   1:  PR[GP1:91,1] = PR[GP1:90,1] + 14.958;
   1:  PR[GP1:91,2] = PR[GP1:90,2] + 47.026;
   1:L PR[91] R[100]mm/sec CNT100;
   1:  PR[GP1:91,1] = PR[GP1:90,1] + 1.682;
   1:  PR[GP1:91,2] = PR[GP1:90,2] + 49.128;
   1:L PR[91] R[100]mm/sec CNT100;
   1:  PR[GP1:91,1] = PR[GP1:90,1] + 0.106;
   1:  PR[GP1:91,2] = PR[GP1:90,2] + 49.323;
   1:L PR[91] R[100]mm/sec CNT100;
   1:  ! -- Layer/Ebene 225 -- !;
   1:  PR[91] = PR[90];
   1:  PR[GP1:91,1] = PR[GP1:90,1] + -0.725;
   1:  PR[GP1:91,2] = PR[GP1:90,2] + 49.220;
   1:  PR[GP1:91,3] = PR[GP1:90,3] + 137.555;
   1:L PR[91] R[100]mm/sec CNT100;
   1:  PR[GP1:91,1] = PR[GP1:90,1] + -14.943;
   1:  PR[GP1:91,2] = PR[GP1:90,2] + 46.968;
   1:L PR[91] R[100]mm/sec CNT100;
   1:  PR[GP1:91,1] = PR[GP1:90,1] + -15.715;
   1:  PR[GP1:91,2] = PR[GP1:90,2] + 46.669;
   1:L PR[91] R[100]mm/sec CNT100;
   1:  PR[GP1:91,1] = PR[GP1:90,1] + -28.542;
   1:  PR[GP1:91,2] = PR[GP1:90,2] + 40.134;
   1:L PR[91] R[100]mm/sec CNT100;
   1:  PR[GP1:91,1] = PR[GP1:90,1] + -29.217;
   1:  PR[GP1:91,2] = PR[GP1:90,2] + 39.656;
   1:L PR[91] R[100]mm/sec CNT100;
   1:  PR[GP1:91,1] = PR[GP1:90,1] + -39.393;
   1:  PR[GP1:91,2] = PR[GP1:90,2] + 29.479;
   1:L PR[91] R[100]mm/sec CNT100;
   1:  PR[GP1:91,1] = PR[GP1:90,1] + -39.995;
   1:  PR[GP1:91,2] = PR[GP1:90,2] + 28.755;
   1:L PR[91] R[100]mm/sec CNT100;
   1:  PR[GP1:91,1] = PR[GP1:90,1] + -46.526;
   1:  PR[GP1:91,2] = PR[GP1:90,2] + 15.936;
   1:L PR[91] R[100]mm/sec CNT100;
   1:  PR[GP1:91,1] = PR[GP1:90,1] + -46.904;
   1:  PR[GP1:91,2] = PR[GP1:90,2] + 15.080;
   1:L PR[91] R[100]mm/sec CNT100;
   1:  PR[GP1:91,1] = PR[GP1:90,1] + -47.036;
   1:  PR[GP1:91,2] = PR[GP1:90,2] + 14.132;
   1:L PR[91] R[100]mm/sec CNT100;
   1:  PR[GP1:91,1] = PR[GP1:90,1] + -49.287;
   1:  PR[GP1:91,2] = PR[GP1:90,2] + -0.078;
   1:L PR[91] R[100]mm/sec CNT100;
   1:  PR[GP1:91,1] = PR[GP1:90,1] + -49.157;
   1:  PR[GP1:91,2] = PR[GP1:90,2] + -1.010;
   1:L PR[91] R[100]mm/sec CNT100;
   1:  PR[GP1:91,1] = PR[GP1:90,1] + -46.906;
   1:  PR[GP1:91,2] = PR[GP1:90,2] + -15.219;
   1:L PR[91] R[100]mm/sec CNT100;
   1:  PR[GP1:91,1] = PR[GP1:90,1] + -46.526;
   1:  PR[GP1:91,2] = PR[GP1:90,2] + -16.080;
   1:L PR[91] R[100]mm/sec CNT100;
   1:  PR[GP1:91,1] = PR[GP1:90,1] + -39.995;
   1:  PR[GP1:91,2] = PR[GP1:90,2] + -28.899;
   1:L PR[91] R[100]mm/sec CNT100;
   1:  PR[GP1:91,1] = PR[GP1:90,1] + -39.393;
   1:  PR[GP1:91,2] = PR[GP1:90,2] + -29.623;
   1:L PR[91] R[100]mm/sec CNT100;
   1:  PR[GP1:91,1] = PR[GP1:90,1] + -29.217;
   1:  PR[GP1:91,2] = PR[GP1:90,2] + -39.800;
   1:L PR[91] R[100]mm/sec CNT100;
   1:  PR[GP1:91,1] = PR[GP1:90,1] + -28.542;
   1:  PR[GP1:91,2] = PR[GP1:90,2] + -40.278;
   1:L PR[91] R[100]mm/sec CNT100;
   1:  PR[GP1:91,1] = PR[GP1:90,1] + -15.715;
   1:  PR[GP1:91,2] = PR[GP1:90,2] + -46.813;
   1:L PR[91] R[100]mm/sec CNT100;
   1:  PR[GP1:91,1] = PR[GP1:90,1] + -14.953;
   1:  PR[GP1:91,2] = PR[GP1:90,2] + -47.109;
   1:L PR[91] R[100]mm/sec CNT100;
   1:  PR[GP1:91,1] = PR[GP1:90,1] + -14.102;
   1:  PR[GP1:91,2] = PR[GP1:90,2] + -47.214;
   1:L PR[91] R[100]mm/sec CNT100;
   1:  PR[GP1:91,1] = PR[GP1:90,1] + 0.117;
   1:  PR[GP1:91,2] = PR[GP1:90,2] + -49.466;
   1:L PR[91] R[100]mm/sec CNT100;
   1:  PR[GP1:91,1] = PR[GP1:90,1] + 0.938;
   1:  PR[GP1:91,2] = PR[GP1:90,2] + -49.364;
   1:L PR[91] R[100]mm/sec CNT100;
   1:  PR[GP1:91,1] = PR[GP1:90,1] + 15.156;
   1:  PR[GP1:91,2] = PR[GP1:90,2] + -47.112;
   1:L PR[91] R[100]mm/sec CNT100;
   1:  PR[GP1:91,1] = PR[GP1:90,1] + 15.928;
   1:  PR[GP1:91,2] = PR[GP1:90,2] + -46.813;
   1:L PR[91] R[100]mm/sec CNT100;
   1:  PR[GP1:91,1] = PR[GP1:90,1] + 28.755;
   1:  PR[GP1:91,2] = PR[GP1:90,2] + -40.278;
   1:L PR[91] R[100]mm/sec CNT100;
   1:  PR[GP1:91,1] = PR[GP1:90,1] + 29.430;
   1:  PR[GP1:91,2] = PR[GP1:90,2] + -39.800;
   1:L PR[91] R[100]mm/sec CNT100;
   1:  PR[GP1:91,1] = PR[GP1:90,1] + 39.607;
   1:  PR[GP1:91,2] = PR[GP1:90,2] + -29.623;
   1:L PR[91] R[100]mm/sec CNT100;
   1:  PR[GP1:91,1] = PR[GP1:90,1] + 40.208;
   1:  PR[GP1:91,2] = PR[GP1:90,2] + -28.899;
   1:L PR[91] R[100]mm/sec CNT100;
   1:  PR[GP1:91,1] = PR[GP1:90,1] + 46.739;
   1:  PR[GP1:91,2] = PR[GP1:90,2] + -16.080;
   1:L PR[91] R[100]mm/sec CNT100;
   1:  PR[GP1:91,1] = PR[GP1:90,1] + 47.117;
   1:  PR[GP1:91,2] = PR[GP1:90,2] + -15.224;
   1:L PR[91] R[100]mm/sec CNT100;
   1:  PR[GP1:91,1] = PR[GP1:90,1] + 47.250;
   1:  PR[GP1:91,2] = PR[GP1:90,2] + -14.275;
   1:L PR[91] R[100]mm/sec CNT100;
   1:  PR[GP1:91,1] = PR[GP1:90,1] + 49.500;
   1:  PR[GP1:91,2] = PR[GP1:90,2] + -0.066;
   1:L PR[91] R[100]mm/sec CNT100;
   1:  PR[GP1:91,1] = PR[GP1:90,1] + 49.370;
   1:  PR[GP1:91,2] = PR[GP1:90,2] + 0.866;
   1:L PR[91] R[100]mm/sec CNT100;
   1:  PR[GP1:91,1] = PR[GP1:90,1] + 47.119;
   1:  PR[GP1:91,2] = PR[GP1:90,2] + 15.075;
   1:L PR[91] R[100]mm/sec CNT100;
   1:  PR[GP1:91,1] = PR[GP1:90,1] + 46.739;
   1:  PR[GP1:91,2] = PR[GP1:90,2] + 15.936;
   1:L PR[91] R[100]mm/sec CNT100;
   1:  PR[GP1:91,1] = PR[GP1:90,1] + 40.208;
   1:  PR[GP1:91,2] = PR[GP1:90,2] + 28.755;
   1:L PR[91] R[100]mm/sec CNT100;
   1:  PR[GP1:91,1] = PR[GP1:90,1] + 39.607;
   1:  PR[GP1:91,2] = PR[GP1:90,2] + 29.479;
   1:L PR[91] R[100]mm/sec CNT100;
   1:  PR[GP1:91,1] = PR[GP1:90,1] + 29.430;
   1:  PR[GP1:91,2] = PR[GP1:90,2] + 39.656;
   1:L PR[91] R[100]mm/sec CNT100;
   1:  PR[GP1:91,1] = PR[GP1:90,1] + 28.755;
   1:  PR[GP1:91,2] = PR[GP1:90,2] + 40.134;
   1:L PR[91] R[100]mm/sec CNT100;
   1:  PR[GP1:91,1] = PR[GP1:90,1] + 15.928;
   1:  PR[GP1:91,2] = PR[GP1:90,2] + 46.669;
   1:L PR[91] R[100]mm/sec CNT100;
   1:  PR[GP1:91,1] = PR[GP1:90,1] + 15.156;
   1:  PR[GP1:91,2] = PR[GP1:90,2] + 46.968;
   1:L PR[91] R[100]mm/sec CNT100;
   1:  PR[GP1:91,1] = PR[GP1:90,1] + 0.938;
   1:  PR[GP1:91,2] = PR[GP1:90,2] + 49.220;
   1:L PR[91] R[100]mm/sec CNT100;
   1:  PR[GP1:91,1] = PR[GP1:90,1] + 0.107;
   1:  PR[GP1:91,2] = PR[GP1:90,2] + 49.323;
   1:L PR[91] R[100]mm/sec CNT100;
   1:  ! -- Layer/Ebene 226 -- !;
   1:  PR[91] = PR[90];
   1:  PR[GP1:91,1] = PR[GP1:90,1] + 0.020;
   1:  PR[GP1:91,2] = PR[GP1:90,2] + 49.313;
   1:  PR[GP1:91,3] = PR[GP1:90,3] + 138.165;
   1:L PR[91] R[100]mm/sec CNT100;
   1:  PR[GP1:91,1] = PR[GP1:90,1] + -15.142;
   1:  PR[GP1:91,2] = PR[GP1:90,2] + 46.911;
   1:L PR[91] R[100]mm/sec CNT100;
   1:  PR[GP1:91,1] = PR[GP1:90,1] + -15.214;
   1:  PR[GP1:91,2] = PR[GP1:90,2] + 46.883;
   1:L PR[91] R[100]mm/sec CNT100;
   1:  PR[GP1:91,1] = PR[GP1:90,1] + -28.891;
   1:  PR[GP1:91,2] = PR[GP1:90,2] + 39.914;
   1:L PR[91] R[100]mm/sec CNT100;
   1:  PR[GP1:91,1] = PR[GP1:90,1] + -28.955;
   1:  PR[GP1:91,2] = PR[GP1:90,2] + 39.870;
   1:L PR[91] R[100]mm/sec CNT100;
   1:  PR[GP1:91,1] = PR[GP1:90,1] + -39.806;
   1:  PR[GP1:91,2] = PR[GP1:90,2] + 29.018;
   1:L PR[91] R[100]mm/sec CNT100;
   1:  PR[GP1:91,1] = PR[GP1:90,1] + -39.869;
   1:  PR[GP1:91,2] = PR[GP1:90,2] + 28.942;
   1:L PR[91] R[100]mm/sec CNT100;
   1:  PR[GP1:91,1] = PR[GP1:90,1] + -46.833;
   1:  PR[GP1:91,2] = PR[GP1:90,2] + 15.273;
   1:L PR[91] R[100]mm/sec CNT100;
   1:  PR[GP1:91,1] = PR[GP1:90,1] + -46.873;
   1:  PR[GP1:91,2] = PR[GP1:90,2] + 15.183;
   1:L PR[91] R[100]mm/sec CNT100;
   1:  PR[GP1:91,1] = PR[GP1:90,1] + -49.287;
   1:  PR[GP1:91,2] = PR[GP1:90,2] + -0.077;
   1:L PR[91] R[100]mm/sec CNT100;
   1:  PR[GP1:91,1] = PR[GP1:90,1] + -49.273;
   1:  PR[GP1:91,2] = PR[GP1:90,2] + -0.176;
   1:L PR[91] R[100]mm/sec CNT100;
   1:  PR[GP1:91,1] = PR[GP1:90,1] + -46.873;
   1:  PR[GP1:91,2] = PR[GP1:90,2] + -15.327;
   1:L PR[91] R[100]mm/sec CNT100;
   1:  PR[GP1:91,1] = PR[GP1:90,1] + -46.833;
   1:  PR[GP1:91,2] = PR[GP1:90,2] + -15.418;
   1:L PR[91] R[100]mm/sec CNT100;
   1:  PR[GP1:91,1] = PR[GP1:90,1] + -39.869;
   1:  PR[GP1:91,2] = PR[GP1:90,2] + -29.086;
   1:L PR[91] R[100]mm/sec CNT100;
   1:  PR[GP1:91,1] = PR[GP1:90,1] + -39.806;
   1:  PR[GP1:91,2] = PR[GP1:90,2] + -29.162;
   1:L PR[91] R[100]mm/sec CNT100;
   1:  PR[GP1:91,1] = PR[GP1:90,1] + -28.955;
   1:  PR[GP1:91,2] = PR[GP1:90,2] + -40.013;
   1:L PR[91] R[100]mm/sec CNT100;
   1:  PR[GP1:91,1] = PR[GP1:90,1] + -28.891;
   1:  PR[GP1:91,2] = PR[GP1:90,2] + -40.058;
   1:L PR[91] R[100]mm/sec CNT100;
   1:  PR[GP1:91,1] = PR[GP1:90,1] + -15.214;
   1:  PR[GP1:91,2] = PR[GP1:90,2] + -47.027;
   1:L PR[91] R[100]mm/sec CNT100;
   1:  PR[GP1:91,1] = PR[GP1:90,1] + -15.142;
   1:  PR[GP1:91,2] = PR[GP1:90,2] + -47.055;
   1:L PR[91] R[100]mm/sec CNT100;
   1:  PR[GP1:91,1] = PR[GP1:90,1] + 0.107;
   1:  PR[GP1:91,2] = PR[GP1:90,2] + -49.465;
   1:L PR[91] R[100]mm/sec CNT100;
   1:  PR[GP1:91,1] = PR[GP1:90,1] + 15.355;
   1:  PR[GP1:91,2] = PR[GP1:90,2] + -47.055;
   1:L PR[91] R[100]mm/sec CNT100;
   1:  PR[GP1:91,1] = PR[GP1:90,1] + 15.427;
   1:  PR[GP1:91,2] = PR[GP1:90,2] + -47.027;
   1:L PR[91] R[100]mm/sec CNT100;
   1:  PR[GP1:91,1] = PR[GP1:90,1] + 29.104;
   1:  PR[GP1:91,2] = PR[GP1:90,2] + -40.058;
   1:L PR[91] R[100]mm/sec CNT100;
   1:  PR[GP1:91,1] = PR[GP1:90,1] + 29.168;
   1:  PR[GP1:91,2] = PR[GP1:90,2] + -40.013;
   1:L PR[91] R[100]mm/sec CNT100;
   1:  PR[GP1:91,1] = PR[GP1:90,1] + 40.019;
   1:  PR[GP1:91,2] = PR[GP1:90,2] + -29.162;
   1:L PR[91] R[100]mm/sec CNT100;
   1:  PR[GP1:91,1] = PR[GP1:90,1] + 40.082;
   1:  PR[GP1:91,2] = PR[GP1:90,2] + -29.086;
   1:L PR[91] R[100]mm/sec CNT100;
   1:  PR[GP1:91,1] = PR[GP1:90,1] + 47.047;
   1:  PR[GP1:91,2] = PR[GP1:90,2] + -15.418;
   1:L PR[91] R[100]mm/sec CNT100;
   1:  PR[GP1:91,1] = PR[GP1:90,1] + 47.087;
   1:  PR[GP1:91,2] = PR[GP1:90,2] + -15.327;
   1:L PR[91] R[100]mm/sec CNT100;
   1:  PR[GP1:91,1] = PR[GP1:90,1] + 49.499;
   1:  PR[GP1:91,2] = PR[GP1:90,2] + -0.072;
   1:L PR[91] R[100]mm/sec CNT100;
   1:  PR[GP1:91,1] = PR[GP1:90,1] + 47.087;
   1:  PR[GP1:91,2] = PR[GP1:90,2] + 15.183;
   1:L PR[91] R[100]mm/sec CNT100;
   1:  PR[GP1:91,1] = PR[GP1:90,1] + 47.047;
   1:  PR[GP1:91,2] = PR[GP1:90,2] + 15.273;
   1:L PR[91] R[100]mm/sec CNT100;
   1:  PR[GP1:91,1] = PR[GP1:90,1] + 40.082;
   1:  PR[GP1:91,2] = PR[GP1:90,2] + 28.942;
   1:L PR[91] R[100]mm/sec CNT100;
   1:  PR[GP1:91,1] = PR[GP1:90,1] + 40.019;
   1:  PR[GP1:91,2] = PR[GP1:90,2] + 29.018;
   1:L PR[91] R[100]mm/sec CNT100;
   1:  PR[GP1:91,1] = PR[GP1:90,1] + 29.168;
   1:  PR[GP1:91,2] = PR[GP1:90,2] + 39.869;
   1:L PR[91] R[100]mm/sec CNT100;
   1:  PR[GP1:91,1] = PR[GP1:90,1] + 29.104;
   1:  PR[GP1:91,2] = PR[GP1:90,2] + 39.914;
   1:L PR[91] R[100]mm/sec CNT100;
   1:  PR[GP1:91,1] = PR[GP1:90,1] + 15.427;
   1:  PR[GP1:91,2] = PR[GP1:90,2] + 46.883;
   1:L PR[91] R[100]mm/sec CNT100;
   1:  PR[GP1:91,1] = PR[GP1:90,1] + 15.355;
   1:  PR[GP1:91,2] = PR[GP1:90,2] + 46.911;
   1:L PR[91] R[100]mm/sec CNT100;
   1:  PR[GP1:91,1] = PR[GP1:90,1] + 0.194;
   1:  PR[GP1:91,2] = PR[GP1:90,2] + 49.313;
   1:L PR[91] R[100]mm/sec CNT100;
   1:  PR[GP1:91,1] = PR[GP1:90,1] + 0.107;
   1:  PR[GP1:91,2] = PR[GP1:90,2] + 49.323;
   1:L PR[91] R[100]mm/sec CNT100;
   1:  PR[GP1:91,1] = PR[GP1:90,1] + 0.020;
   1:  PR[GP1:91,2] = PR[GP1:90,2] + 49.313;
   1:L PR[91] R[100]mm/sec CNT100;
   1:  PR[GP1:91,1] = PR[GP1:90,1] + -15.142;
   1:  PR[GP1:91,2] = PR[GP1:90,2] + 46.911;
   1:L PR[91] R[100]mm/sec CNT100;
   1:  PR[GP1:91,1] = PR[GP1:90,1] + -15.214;
   1:  PR[GP1:91,2] = PR[GP1:90,2] + 46.883;
   1:L PR[91] R[100]mm/sec CNT100;
   1:  PR[GP1:91,1] = PR[GP1:90,1] + -28.891;
   1:  PR[GP1:91,2] = PR[GP1:90,2] + 39.914;
   1:L PR[91] R[100]mm/sec CNT100;
   1:  PR[GP1:91,1] = PR[GP1:90,1] + -28.955;
   1:  PR[GP1:91,2] = PR[GP1:90,2] + 39.870;
   1:L PR[91] R[100]mm/sec CNT100;
   1:  PR[GP1:91,1] = PR[GP1:90,1] + -39.806;
   1:  PR[GP1:91,2] = PR[GP1:90,2] + 29.018;
   1:L PR[91] R[100]mm/sec CNT100;
   1:  PR[GP1:91,1] = PR[GP1:90,1] + -39.869;
   1:  PR[GP1:91,2] = PR[GP1:90,2] + 28.942;
   1:L PR[91] R[100]mm/sec CNT100;
   1:  PR[GP1:91,1] = PR[GP1:90,1] + -46.833;
   1:  PR[GP1:91,2] = PR[GP1:90,2] + 15.273;
   1:L PR[91] R[100]mm/sec CNT100;
   1:  PR[GP1:91,1] = PR[GP1:90,1] + -46.873;
   1:  PR[GP1:91,2] = PR[GP1:90,2] + 15.183;
   1:L PR[91] R[100]mm/sec CNT100;
   1:  PR[GP1:91,1] = PR[GP1:90,1] + -49.287;
   1:  PR[GP1:91,2] = PR[GP1:90,2] + -0.077;
   1:L PR[91] R[100]mm/sec CNT100;
   1:  PR[GP1:91,1] = PR[GP1:90,1] + -49.273;
   1:  PR[GP1:91,2] = PR[GP1:90,2] + -0.176;
   1:L PR[91] R[100]mm/sec CNT100;
   1:  PR[GP1:91,1] = PR[GP1:90,1] + -46.873;
   1:  PR[GP1:91,2] = PR[GP1:90,2] + -15.327;
   1:L PR[91] R[100]mm/sec CNT100;
   1:  PR[GP1:91,1] = PR[GP1:90,1] + -46.833;
   1:  PR[GP1:91,2] = PR[GP1:90,2] + -15.418;
   1:L PR[91] R[100]mm/sec CNT100;
   1:  PR[GP1:91,1] = PR[GP1:90,1] + -39.869;
   1:  PR[GP1:91,2] = PR[GP1:90,2] + -29.086;
   1:L PR[91] R[100]mm/sec CNT100;
   1:  PR[GP1:91,1] = PR[GP1:90,1] + -39.806;
   1:  PR[GP1:91,2] = PR[GP1:90,2] + -29.162;
   1:L PR[91] R[100]mm/sec CNT100;
   1:  PR[GP1:91,1] = PR[GP1:90,1] + -28.955;
   1:  PR[GP1:91,2] = PR[GP1:90,2] + -40.013;
   1:L PR[91] R[100]mm/sec CNT100;
   1:  PR[GP1:91,1] = PR[GP1:90,1] + -28.891;
   1:  PR[GP1:91,2] = PR[GP1:90,2] + -40.058;
   1:L PR[91] R[100]mm/sec CNT100;
   1:  PR[GP1:91,1] = PR[GP1:90,1] + -15.214;
   1:  PR[GP1:91,2] = PR[GP1:90,2] + -47.027;
   1:L PR[91] R[100]mm/sec CNT100;
   1:  PR[GP1:91,1] = PR[GP1:90,1] + -15.142;
   1:  PR[GP1:91,2] = PR[GP1:90,2] + -47.055;
   1:L PR[91] R[100]mm/sec CNT100;
   1:  PR[GP1:91,1] = PR[GP1:90,1] + 0.107;
   1:  PR[GP1:91,2] = PR[GP1:90,2] + -49.465;
   1:L PR[91] R[100]mm/sec CNT100;
   1:  PR[GP1:91,1] = PR[GP1:90,1] + 15.355;
   1:  PR[GP1:91,2] = PR[GP1:90,2] + -47.055;
   1:L PR[91] R[100]mm/sec CNT100;
   1:  PR[GP1:91,1] = PR[GP1:90,1] + 15.427;
   1:  PR[GP1:91,2] = PR[GP1:90,2] + -47.027;
   1:L PR[91] R[100]mm/sec CNT100;
   1:  PR[GP1:91,1] = PR[GP1:90,1] + 29.104;
   1:  PR[GP1:91,2] = PR[GP1:90,2] + -40.058;
   1:L PR[91] R[100]mm/sec CNT100;
   1:  PR[GP1:91,1] = PR[GP1:90,1] + 29.168;
   1:  PR[GP1:91,2] = PR[GP1:90,2] + -40.013;
   1:L PR[91] R[100]mm/sec CNT100;
   1:  PR[GP1:91,1] = PR[GP1:90,1] + 40.019;
   1:  PR[GP1:91,2] = PR[GP1:90,2] + -29.162;
   1:L PR[91] R[100]mm/sec CNT100;
   1:  PR[GP1:91,1] = PR[GP1:90,1] + 40.082;
   1:  PR[GP1:91,2] = PR[GP1:90,2] + -29.086;
   1:L PR[91] R[100]mm/sec CNT100;
   1:  PR[GP1:91,1] = PR[GP1:90,1] + 47.047;
   1:  PR[GP1:91,2] = PR[GP1:90,2] + -15.418;
   1:L PR[91] R[100]mm/sec CNT100;
   1:  PR[GP1:91,1] = PR[GP1:90,1] + 47.087;
   1:  PR[GP1:91,2] = PR[GP1:90,2] + -15.327;
   1:L PR[91] R[100]mm/sec CNT100;
   1:  PR[GP1:91,1] = PR[GP1:90,1] + 49.499;
   1:  PR[GP1:91,2] = PR[GP1:90,2] + -0.072;
   1:L PR[91] R[100]mm/sec CNT100;
   1:  PR[GP1:91,1] = PR[GP1:90,1] + 47.087;
   1:  PR[GP1:91,2] = PR[GP1:90,2] + 15.183;
   1:L PR[91] R[100]mm/sec CNT100;
   1:  PR[GP1:91,1] = PR[GP1:90,1] + 47.047;
   1:  PR[GP1:91,2] = PR[GP1:90,2] + 15.273;
   1:L PR[91] R[100]mm/sec CNT100;
   1:  PR[GP1:91,1] = PR[GP1:90,1] + 40.082;
   1:  PR[GP1:91,2] = PR[GP1:90,2] + 28.942;
   1:L PR[91] R[100]mm/sec CNT100;
   1:  PR[GP1:91,1] = PR[GP1:90,1] + 40.019;
   1:  PR[GP1:91,2] = PR[GP1:90,2] + 29.018;
   1:L PR[91] R[100]mm/sec CNT100;
   1:  PR[GP1:91,1] = PR[GP1:90,1] + 29.168;
   1:  PR[GP1:91,2] = PR[GP1:90,2] + 39.869;
   1:L PR[91] R[100]mm/sec CNT100;
   1:  PR[GP1:91,1] = PR[GP1:90,1] + 29.104;
   1:  PR[GP1:91,2] = PR[GP1:90,2] + 39.914;
   1:L PR[91] R[100]mm/sec CNT100;
   1:  PR[GP1:91,1] = PR[GP1:90,1] + 15.427;
   1:  PR[GP1:91,2] = PR[GP1:90,2] + 46.883;
   1:L PR[91] R[100]mm/sec CNT100;
   1:  PR[GP1:91,1] = PR[GP1:90,1] + 15.355;
   1:  PR[GP1:91,2] = PR[GP1:90,2] + 46.911;
   1:L PR[91] R[100]mm/sec CNT100;
   1:  PR[GP1:91,1] = PR[GP1:90,1] + 0.194;
   1:  PR[GP1:91,2] = PR[GP1:90,2] + 49.313;
   1:L PR[91] R[100]mm/sec CNT100;
   1:  PR[GP1:91,1] = PR[GP1:90,1] + 0.107;
   1:  PR[GP1:91,2] = PR[GP1:90,2] + 49.323;
   1:L PR[91] R[100]mm/sec CNT100 TB   .50sec,CALL END_PUD;
   1:  DO[117:Laser Start]=OFF;
   1:  !Sicherheitspunkt!;
   1:  PR[92] = PR[91];
   1:  PR[92] = PR[GP1:92,3] + 50;
   1:J PR[92];
   1:  WAIT   5.00(sec);
   1:  DO[119:Gas]=OFF;
   1:  CALL HOME_ALL;
/POS
/END
